// TIA Portal V16 export
// export: Created 2022-07-21T09:35:19.5340597Z, ExportSetting WithDefaults, DisplayName Totally Integrated Automation Portal, DisplayVersion V16 Update 4, DisplayName TIA Portal Version Control Interface, DisplayVersion V16 Update 2, DisplayName TIA Portal Openness, DisplayVersion V16 Update 4, DisplayName SINAMICS Startdrive Advanced, DisplayVersion V16 Update 5, DisplayName SINAMICS Startdrive G130, G150, S120, S150, SINAMICS MV, S210, DisplayVersion V16 Update 5, DisplayName SINAMICS Startdrive G110M, G120, G120C, G120D, G120P, G115D, DisplayVersion V16 Update 5, DisplayName STEP 7 Professional, DisplayVersion V16 Update 4, DisplayName STEP 7 Safety, DisplayVersion V16, DisplayName WinCC Advanced, DisplayVersion V16 Update 4
FUNCTION_BLOCK "fbCoolingZoneCoding"   // FB40, LAD
TITLE = Cooling - position coding / Suszarka - kodowanie pozycji
{ S7_Optimized_Access := 'TRUE' }
VERSION : 0.1
// stored: AutoNumber true, IsIECCheckEnabled false, IsRetainMemResEnabled false, MemoryReserve 100, SetENOAutomatically false, UDAEnableTagReadback false
   VAR_INPUT
      in : Byte;
   END_VAR
   VAR_IN_OUT
      io : "typeRotaryDriveSts";
   END_VAR
   VAR
      sFieldSensors0OUT { ExternalAccessible := 'False'; ExternalVisible := 'False'; ExternalWritable := 'False'} : Struct
         home { ExternalAccessible := 'False'; ExternalVisible := 'False'; ExternalWritable := 'False'} : Bool;
         work { ExternalAccessible := 'False'; ExternalVisible := 'False'; ExternalWritable := 'False'} : Bool;
         pos { ExternalAccessible := 'False'; ExternalVisible := 'False'; ExternalWritable := 'False'} : Bool;
      END_STRUCT;
      sFieldSensors1OUT { ExternalAccessible := 'False'; ExternalVisible := 'False'; ExternalWritable := 'False'} : Struct
         home { ExternalAccessible := 'False'; ExternalVisible := 'False'; ExternalWritable := 'False'} : Bool;
         work { ExternalAccessible := 'False'; ExternalVisible := 'False'; ExternalWritable := 'False'} : Bool;
         pos { ExternalAccessible := 'False'; ExternalVisible := 'False'; ExternalWritable := 'False'} : Bool;
      END_STRUCT;
      sFieldSensors2OUT { ExternalAccessible := 'False'; ExternalVisible := 'False'; ExternalWritable := 'False'} : Struct
         home { ExternalAccessible := 'False'; ExternalVisible := 'False'; ExternalWritable := 'False'} : Bool;
         work { ExternalAccessible := 'False'; ExternalVisible := 'False'; ExternalWritable := 'False'} : Bool;
         pos { ExternalAccessible := 'False'; ExternalVisible := 'False'; ExternalWritable := 'False'} : Bool;
      END_STRUCT;
      sFieldSensors3OUT { ExternalAccessible := 'False'; ExternalVisible := 'False'; ExternalWritable := 'False'} : Struct
         home { ExternalAccessible := 'False'; ExternalVisible := 'False'; ExternalWritable := 'False'} : Bool;
         work { ExternalAccessible := 'False'; ExternalVisible := 'False'; ExternalWritable := 'False'} : Bool;
         pos { ExternalAccessible := 'False'; ExternalVisible := 'False'; ExternalWritable := 'False'} : Bool;
      END_STRUCT;
      sFieldSensors4OUT { ExternalAccessible := 'False'; ExternalVisible := 'False'; ExternalWritable := 'False'} : Struct
         home { ExternalAccessible := 'False'; ExternalVisible := 'False'; ExternalWritable := 'False'} : Bool;
         work { ExternalAccessible := 'False'; ExternalVisible := 'False'; ExternalWritable := 'False'} : Bool;
         pos { ExternalAccessible := 'False'; ExternalVisible := 'False'; ExternalWritable := 'False'} : Bool;
      END_STRUCT;
      sNoCoding { ExternalAccessible := 'False'; ExternalVisible := 'False'; ExternalWritable := 'False'} : Bool;
   END_VAR
   VAR_TEMP
      tTT1Coding : Byte;
      tFieldSensors0IN : Struct
         home : Bool;
         work : Bool;
         pos : Bool;
      END_STRUCT;
      tFieldSensors1IN : Struct
         home : Bool;
         work : Bool;
         pos : Bool;
      END_STRUCT;
      tFieldSensors2IN : Struct
         home : Bool;
         work : Bool;
         pos : Bool;
      END_STRUCT;
      tFieldSensors3IN : Struct
         home : Bool;
         work : Bool;
         pos : Bool;
      END_STRUCT;
      tFieldSensors4IN : Struct
         home : Bool;
         work : Bool;
         pos : Bool;
      END_STRUCT;
   END_VAR
BEGIN

REGION Network 1: Position coding / Kodowanie pozycji
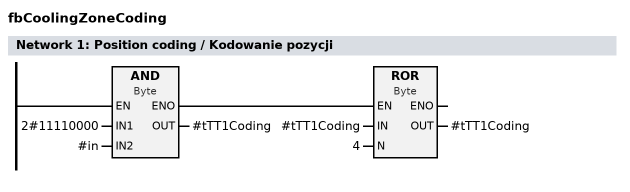
   #tTT1Coding := 2#11110000 AND #in;
   #tTT1Coding := ROR(IN := #tTT1Coding, N := 4);
END_REGION

REGION Network 2 (SCL): Copy inputs / Przepisanie wejść

   IF #io.inPosition THEN
       CASE #tTT1Coding OF
           1:
               #io.position := 1;
           2:
               #io.position := 2;
           3:
               #io.position := 3;
           4:
               #io.position := 4;
           6:
               #io.position := 5;
           7:
               #io.position := 6;
           8:
               #io.position := 7;
           11:
               #io.position := 8;
           12:
               #io.position := 9;
           13:
               #io.position := 10;
           14:
               #io.position := 11;
           15:
               #io.position := 12;

       END_CASE;
   ELSE
       #io.position := 0;
   END_IF;
END_REGION
END_FUNCTION_BLOCK
